INTERFACE I_SeasonControl EXTENDS __SYSTEM.IQueryInterface

PROPERTY StateAutumn : I_State
GET
END_GET
END_PROPERTY

PROPERTY StateSpring : I_State
GET
END_GET
END_PROPERTY

PROPERTY StateSummer : I_State
GET
END_GET
END_PROPERTY

PROPERTY StateWinter : I_State
GET
END_GET
END_PROPERTY

END_INTERFACE

(* stored: Version 1.1.0.1, ProductVersion 3.1.4024.12
   Itf I_SeasonControl: Id {12974377-d928-4e78-b12c-77b03d643d5c}
   Property StateAutumn: Id {2e1533d9-9e35-4e7a-bef3-18312995aa00}
   Get Get: Id {ae790c19-22df-4b2f-bee9-b3ec99e60d90}
   Property StateSpring: Id {d4526630-5bb5-4c74-ba2d-0851a0363c97}
   Get Get: Id {c4de62ea-0512-4b4b-8887-ecc515cbd083}
   Property StateSummer: Id {85916644-f4d4-4b03-9949-acb890eef573}
   Get Get: Id {f6d38104-5be9-42f4-bb78-7163041ba3e4}
   Property StateWinter: Id {f73bcb29-6f11-4372-b4ba-bb5bc1ebb938}
   Get Get: Id {7a907ffa-70f3-40a4-9b52-41c3e54c7ec6} *)
